{attribute 'linkalways'} 
{attribute 'no_explicit_call' := 'This FB is a CLASS and must be accessed using methods or properties'}
{attribute 'enable_dynamic_creation'}
FUNCTION_BLOCK Node_F_VN_ExportImageSize EXTENDS VisionNode
VAR
    ipImage : _ITcVnImage;
    nBufferSize : _ULINT(0);
    hrPrev : _HRESULT(S_OK);
	hresult : _HRESULT(S_OK);
END_VAR

METHOD PUBLIC  Clone : I_Node
VAR
	pNode : POINTER TO Node_F_VN_ExportImageSize;
END_VAR
pNode := __NEW(Node_F_VN_ExportImageSize);
Clone := pNode^;
END_METHOD

METHOD FB_init : BOOL
VAR_INPUT
	bInitRetains : BOOL; // if TRUE, the retain variables are initialized (warm start / cold start)
	bInCopyCode : BOOL;  // if TRUE, the instance afterwards gets moved into the copy code (online change)
END_VAR
AddInput('ipImage', ipImage);
AddInput('hrPrev', hrPrev);
AddOutput('nBufferSize', nBufferSize);
AddOutput('hresult',hresult);
END_METHOD

METHOD PROTECTED  OnExecute : HRESULT
hresult.Value := F_VN_ExportImageSize(
    ipImage := ipImage.Value,
    nBufferSize := nBufferSize.Value,
	hrPrev:= hrPrev.Value);
END_METHOD

METHOD PUBLIC PreExecutionCheck
VAR_INPUT
	Check : I_PreExecutionChecks;
END_VAR
Check.IsTrue(ipImage.IsValid, 'ipImage must contain an image');
END_METHOD

END_FUNCTION_BLOCK

(* stored: Version 1.1.0.1, ProductVersion 3.1.4024.13
   POU Node_F_VN_ExportImageSize: Id {1224ce58-81d9-0b19-1581-09f80140ed3a}, SpecialFunc None
   Folder Constructor: Id {bbc599cc-193d-070f-2ea1-542117749be5}
   Method Clone: Id {a444706e-3685-047c-3c2b-db7aa6c50552}
   Method FB_init: Id {8a9ee821-a640-0ce9-28f4-ed2d7fd3ca71}
   Method OnExecute: Id {282bf096-6fa5-097e-238b-8147e8e1265b}
   Method PreExecutionCheck: Id {da2548d7-9377-0fe6-3e00-1cfd61763057} *)
